// Examples of groups.
FUNCTION_BLOCK FB_Ref_Groups EXTENDS FB_BA_View
VAR
	{region 'Analog'}
		A							: FB_BA_View := (
										iParent							:= THIS^,
										sDescription					:= '{Analog objects}'
									);
				                    
			GrpAV1					: FB_BA_AV := (
										iParent							:= A,
										eUnit							:= E_BA_Unit.eOther_NoUnits,
										nEventClassID					:= 11,
										bEnPgm							:= TRUE,
										fValPgm							:= 10
									);
			GrpAV2					: FB_BA_AV := (
										iParent							:= A,
										eUnit							:= E_BA_Unit.eOther_NoUnits,
										nEventClassID					:= 11,
										bEnPgm							:= TRUE,
										fValPgm							:= 15
									);
			GrpAVOp1				: FB_BA_AV_Op := (
										iParent							:= A,
										eUnit							:= E_BA_Unit.eTemperature_DegreesCelsius,
										fValueRm						:= 20
									);
			GrpAVOp2				: FB_BA_AV_Op := (
										iParent							:= A,
										eUnit							:= E_BA_Unit.eTemperature_DegreesCelsius,
										fValueRm						:= 25
									);
										 
			// Intention:			Eigenständige Gruppe (Ohne Achsen-Zugehörigkeit)
			Group_AVMin				: FB_BA_Group_AVal := (
										eCalcMode						:= E_BA_AValCalcMode.eMin,
										iReference						:= [ GrpAV1, GrpAV2, GrpAVOp1, GrpAVOp2 ]
									);
			Group_AVMax				: FB_BA_Group_AVal := (
										eCalcMode						:= E_BA_AValCalcMode.eMax,
										iReference						:= [ GrpAV1, GrpAV2, GrpAVOp1, GrpAVOp2 ]
									);
			Group_AVAvg				: FB_BA_Group_AVal := (
										eCalcMode						:= E_BA_AValCalcMode.eAverage,
										iReference						:= [ GrpAV1, GrpAV2, GrpAVOp1, GrpAVOp2 ]
									);
	{endregion}
END_VAR

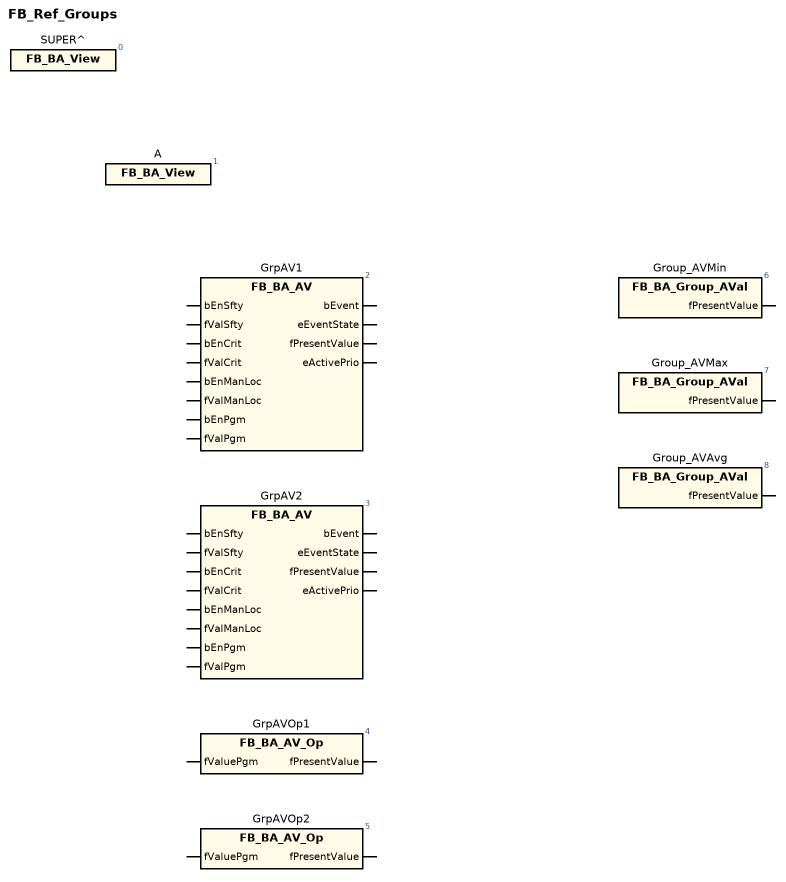
SUPER^(); // FB_BA_View
A(); // FB_BA_View
GrpAV1(); // FB_BA_AV
GrpAV2(); // FB_BA_AV
GrpAVOp1(); // FB_BA_AV_Op
GrpAVOp2(); // FB_BA_AV_Op
Group_AVMin(); // FB_BA_Group_AVal
Group_AVMax(); // FB_BA_Group_AVal
Group_AVAvg(); // FB_BA_Group_AVal

END_FUNCTION_BLOCK

(* stored: Version 1.1.0.1, ProductVersion 3.1.4024.5
   POU FB_Ref_Groups: Id {9f032fce-b80b-4d6c-8d01-f421abd175da}, SpecialFunc None *)
